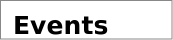
VISUALIZATION VISU_HMI_EVENTS  // 173x40
    Label (10,10 163x30), "Events"
END_VISUALIZATION

(* stored: Version 1.1.0.1, ProductVersion 3.1.4024.14
   Visu VISU_HMI_EVENTS: Id {e808af8b-ba4d-4433-a35f-a0bdb8d442cd} *)
